// TIA Portal V17 export
// export: Created 2024-06-16T17:47:39.2675284Z, ExportSetting WithDefaults, DisplayName Totally Integrated Automation Portal, DisplayVersion V17, DisplayName TIA Portal Openness, DisplayVersion V17, DisplayName TIA Portal Version Control Interface, DisplayVersion V17, DisplayName STEP 7 Professional, DisplayVersion V17, DisplayName STEP 7 Safety, DisplayVersion V17, DisplayName WinCC Professional, DisplayVersion V17
VAR_GLOBAL   // PLC tag table "St1_In"
   IO_Pinces_Ouvert AT %I1.0 : Bool;   // Pinces de préhension Z : Ouverte
   IO_Pinces_Fermee AT %I1.1 : Bool;   // Pinces de préhension Z : Fermée
   IO_Cpt_C1 AT %I1.2 : Bool;   // Présence pile devant capteur Chargement AR : C1
   IO_Cpt_C2 AT %I1.3 : Bool;   // Présence pile devant capteur Chargement AR : C2
   IO_Cpt_C3 AT %I1.4 : Bool;   // Présence pile devant capteur Chargement AV : C3
   IO_Cpt_C4 AT %I1.5 : Bool;   // Présence pile devant capteur Chargement AV : C4
   IO_Cpt_C5 AT %I1.6 : Bool;   // Présence pile devant capteur Dépilement : C5
   IO_Cpt_C6 AT %I1.7 : Bool;   // Détection collage barquette Dépilement : C6
   IO_Cpt_C7 AT %I2.0 : Bool;   // Détection collage barquette Dépilement : C7
END_VAR
